PROGRAM F00_Safety_Signals
VAR
	fbPSR_IsReset				: FB_IO2_SingleInputCtrl;		(**)
	fbPSR_OK					: FB_IO2_SingleInputCtrl;		(**)
	fbEmergencyStop			: FB_IO2_SingleInputCtrl;		(**)
	fbEmergencyCircuit		: FB_IO2_SingleInputCtrl;		(**)
	fbMotorInverterOK			: FB_IO2_SingleInputCtrl;		(**)
	fbGuardDoorOK			: FB_IO2_SingleInputCtrl;		(**)

END_VAR

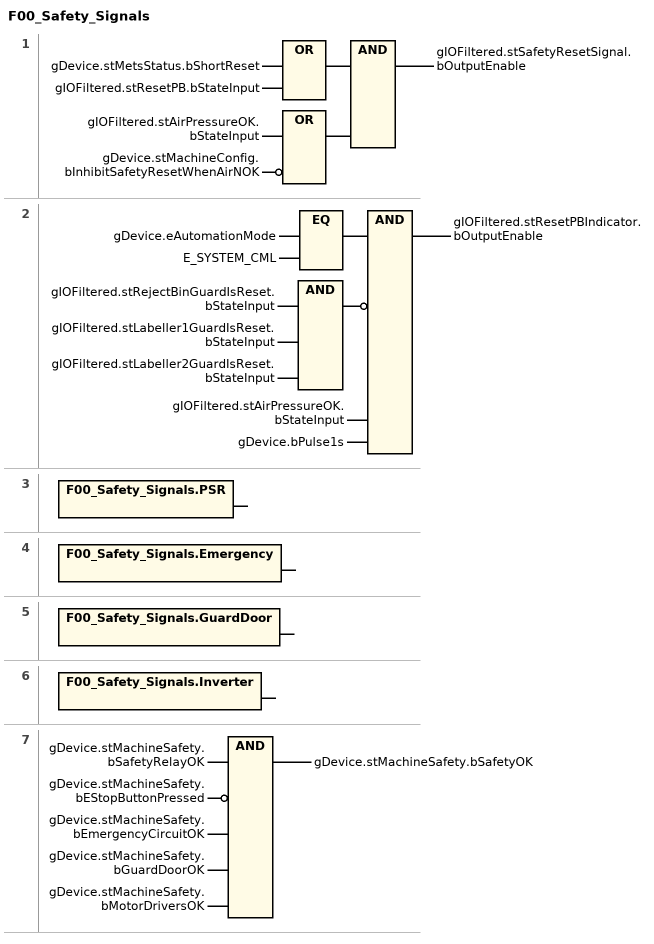
// NETWORK 1
gIOFiltered.stSafetyResetSignal.bOutputEnable := (gDevice.stMetsStatus.bShortReset OR gIOFiltered.stResetPB.bStateInput) AND (gIOFiltered.stAirPressureOK.bStateInput OR NOT gDevice.stMachineConfig.bInhibitSafetyResetWhenAirNOK);

// NETWORK 2
gIOFiltered.stResetPBIndicator.bOutputEnable := gDevice.eAutomationMode = E_SYSTEM_CML AND NOT (gIOFiltered.stRejectBinGuardIsReset.bStateInput AND gIOFiltered.stLabeller1GuardIsReset.bStateInput AND gIOFiltered.stLabeller2GuardIsReset.bStateInput) AND gIOFiltered.stAirPressureOK.bStateInput AND gDevice.bPulse1s;

// NETWORK 3
F00_Safety_Signals.PSR();

// NETWORK 4
F00_Safety_Signals.Emergency();

// NETWORK 5
F00_Safety_Signals.GuardDoor();

// NETWORK 6
F00_Safety_Signals.Inverter();

// NETWORK 7
gDevice.stMachineSafety.bSafetyOK := gDevice.stMachineSafety.bSafetyRelayOK AND NOT gDevice.stMachineSafety.bEStopButtonPressed AND gDevice.stMachineSafety.bEmergencyCircuitOK AND gDevice.stMachineSafety.bGuardDoorOK AND gDevice.stMachineSafety.bMotorDriversOK;

ACTION Emergency:
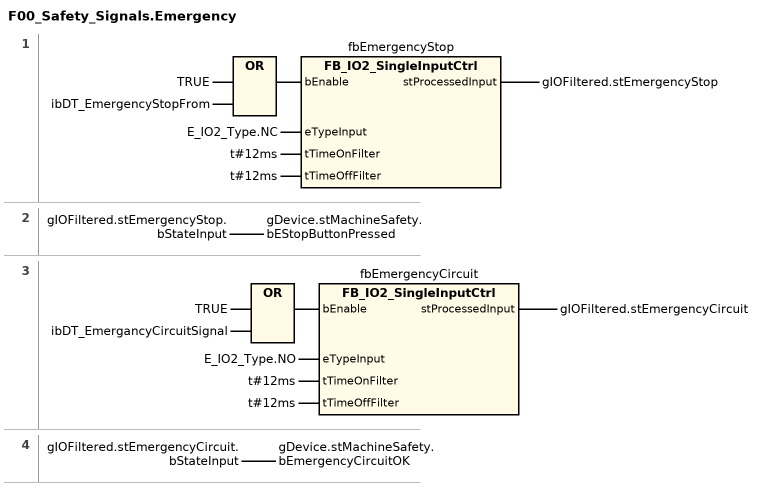
// NETWORK 1
fbEmergencyStop(
    bEnable := TRUE OR ibDT_EmergencyStopFrom,
    eTypeInput := E_IO2_Type.NC,
    tTimeOnFilter := t#12ms,
    tTimeOffFilter := t#12ms); // FB_IO2_SingleInputCtrl
gIOFiltered.stEmergencyStop := fbEmergencyStop.stProcessedInput;

// NETWORK 2
gDevice.stMachineSafety.bEStopButtonPressed := gIOFiltered.stEmergencyStop.bStateInput;

// NETWORK 3
fbEmergencyCircuit(
    bEnable := TRUE OR ibDT_EmergancyCircuitSignal,
    eTypeInput := E_IO2_Type.NO,
    tTimeOnFilter := t#12ms,
    tTimeOffFilter := t#12ms); // FB_IO2_SingleInputCtrl
gIOFiltered.stEmergencyCircuit := fbEmergencyCircuit.stProcessedInput;

// NETWORK 4
gDevice.stMachineSafety.bEmergencyCircuitOK := gIOFiltered.stEmergencyCircuit.bStateInput;
END_ACTION

ACTION GuardDoor:
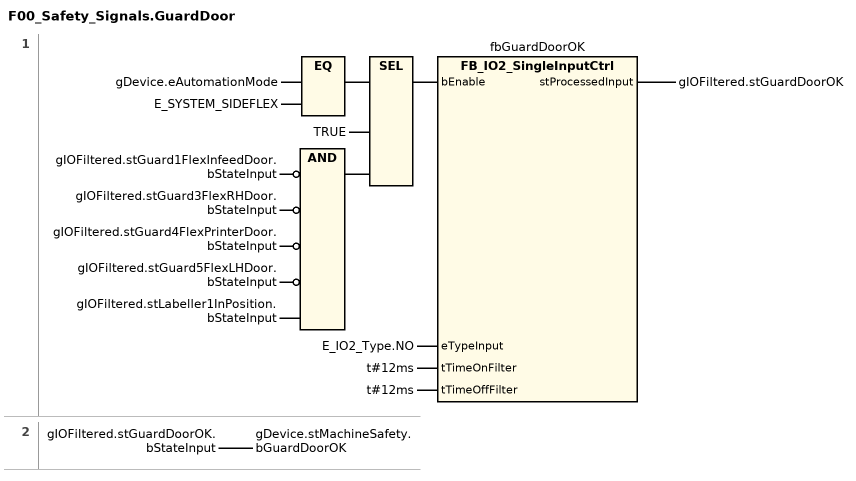
// NETWORK 1
fbGuardDoorOK(
    bEnable := SEL(gDevice.eAutomationMode = E_SYSTEM_SIDEFLEX, TRUE, NOT gIOFiltered.stGuard1FlexInfeedDoor.bStateInput AND NOT gIOFiltered.stGuard3FlexRHDoor.bStateInput AND NOT gIOFiltered.stGuard4FlexPrinterDoor.bStateInput AND NOT gIOFiltered.stGuard5FlexLHDoor.bStateInput AND gIOFiltered.stLabeller1InPosition.bStateInput),
    eTypeInput := E_IO2_Type.NO,
    tTimeOnFilter := t#12ms,
    tTimeOffFilter := t#12ms); // FB_IO2_SingleInputCtrl
gIOFiltered.stGuardDoorOK := fbGuardDoorOK.stProcessedInput;

// NETWORK 2
gDevice.stMachineSafety.bGuardDoorOK := gIOFiltered.stGuardDoorOK.bStateInput;
END_ACTION

ACTION Inverter:
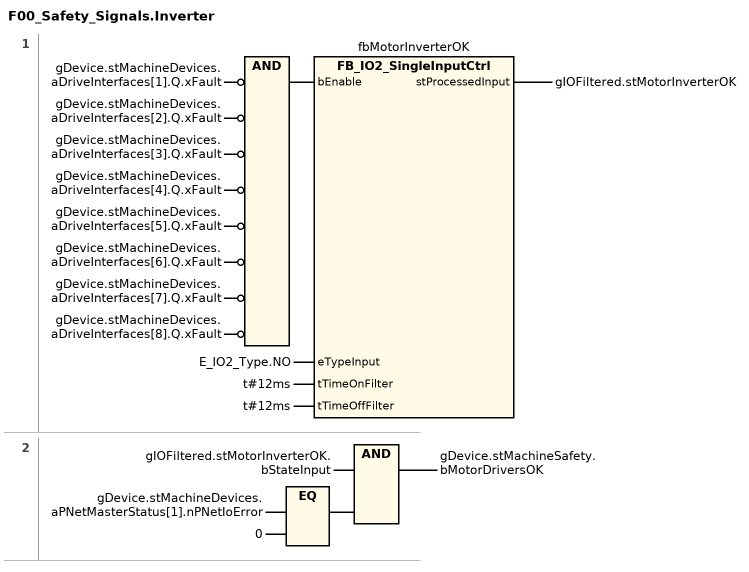
// NETWORK 1
fbMotorInverterOK(
    bEnable := NOT gDevice.stMachineDevices.aDriveInterfaces[1].Q.xFault AND NOT gDevice.stMachineDevices.aDriveInterfaces[2].Q.xFault AND NOT gDevice.stMachineDevices.aDriveInterfaces[3].Q.xFault AND NOT gDevice.stMachineDevices.aDriveInterfaces[4].Q.xFault AND NOT gDevice.stMachineDevices.aDriveInterfaces[5].Q.xFault AND NOT gDevice.stMachineDevices.aDriveInterfaces[6].Q.xFault AND NOT gDevice.stMachineDevices.aDriveInterfaces[7].Q.xFault AND NOT gDevice.stMachineDevices.aDriveInterfaces[8].Q.xFault,
    eTypeInput := E_IO2_Type.NO,
    tTimeOnFilter := t#12ms,
    tTimeOffFilter := t#12ms); // FB_IO2_SingleInputCtrl
gIOFiltered.stMotorInverterOK := fbMotorInverterOK.stProcessedInput;

// NETWORK 2
gDevice.stMachineSafety.bMotorDriversOK := gIOFiltered.stMotorInverterOK.bStateInput AND gDevice.stMachineDevices.aPNetMasterStatus[1].nPNetIoError = 0;
END_ACTION

ACTION PSR:
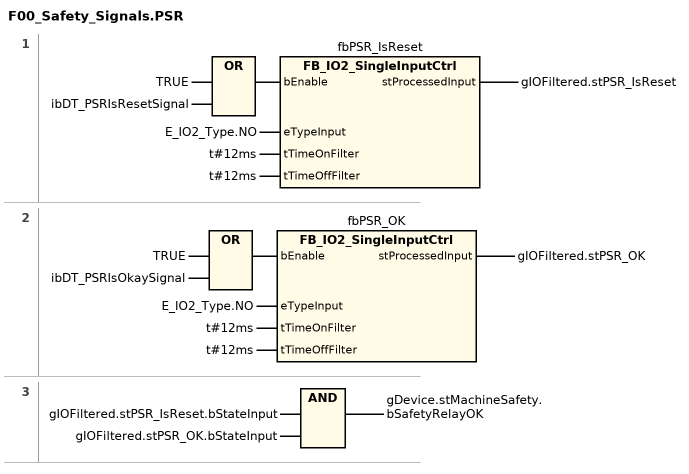
// NETWORK 1
fbPSR_IsReset(
    bEnable := TRUE OR ibDT_PSRIsResetSignal,
    eTypeInput := E_IO2_Type.NO,
    tTimeOnFilter := t#12ms,
    tTimeOffFilter := t#12ms); // FB_IO2_SingleInputCtrl
gIOFiltered.stPSR_IsReset := fbPSR_IsReset.stProcessedInput;

// NETWORK 2
fbPSR_OK(
    bEnable := TRUE OR ibDT_PSRIsOkaySignal,
    eTypeInput := E_IO2_Type.NO,
    tTimeOnFilter := t#12ms,
    tTimeOffFilter := t#12ms); // FB_IO2_SingleInputCtrl
gIOFiltered.stPSR_OK := fbPSR_OK.stProcessedInput;

// NETWORK 3
gDevice.stMachineSafety.bSafetyRelayOK := gIOFiltered.stPSR_IsReset.bStateInput AND gIOFiltered.stPSR_OK.bStateInput;
END_ACTION

END_PROGRAM

(* stored: Version 1.1.0.1
   POU F00_Safety_Signals: Id {3276de5e-d54d-40e4-adbe-c200cb057b8f}, SpecialFunc None
   Action Emergency: Id {9a01ebb7-0361-4b14-91f4-d20d03a054f1}
   Action GuardDoor: Id {5cba5ba4-6632-4c8b-b67f-a521b865066c}
   Action Inverter: Id {f6b19e95-9a9a-4606-a139-4019be2126eb}
   Action PSR: Id {ed09a51d-e939-4022-800c-4a7d40bd6529} *)
